PROGRAM pTimer
VAR
	timer : TON;
END_VAR

timer(IN := TRUE, PT := T#5S);
IF timer.Q THEN
	PeriodicMesure();
	timer(IN := NOT PeriodicMesure.isfinished());
END_IF

END_PROGRAM

(* stored: Version 1.1.0.1, ProductVersion 3.1.4024.12
   POU pTimer: Id {8fcbf0f7-6c45-4986-b034-e15f9132d3c4}, SpecialFunc None *)
